// TIA Portal project "2022.09.06-步进电机仿真" (V17)

(* hardware
DEVICE "HMI_1"  KTP700 Basic PN
   slot 0: "HMI_1"  KTP700 Basic PN  6AV2 123-2GB03-0AX0  15.1.0.0
   slot 1: "HMI_RT_1"  KTP700 Basic PN  6AV2 123-2GB03-0AX0  15.1.0.0
   slot 5: "HMI_1.IE_CP_1"  PROFINET Interface  15.0.1.0
      slot 1: "PROFINET Interface_1"  PROFINET Interface
         slot 1: "Port_1"  Port
DEVICE "S7-1200 station_1"  S7-1200 Station
   slot 0: "Rack_0"  S7-1200 Rack  Rack  V1.0
   slot 1: "PLC_1"  CPU 1214C DC/DC/DC  6ES7 214-1AG40-0XB0  V4.2
*)

// ===== PLC "PLC_1"  CPU 1214C DC/DC/DC =====

VAR_GLOBAL   // PLC tag table "默认变量表"
   "反转按钮" AT %I0.1 : Bool;
   "正转KA1" AT %Q0.0 : Bool;
   "反转KA2" AT %Q0.1 : Bool;
   "停止按钮" AT %I0.2 : Bool;
   "正转按钮" AT %I0.0 : Bool;
   "正转按钮触摸屏" AT %M0.0 : Bool;
   "反转按钮触摸屏" AT %M0.1 : Bool;
   "停止按钮触摸屏" AT %M0.2 : Bool;
   "正转触摸屏指示灯" AT %M1.0 : Bool;
   "反转触摸屏指示灯" AT %M1.1 : Bool;
   "电动机转速" AT %MD20 : DWord;
END_VAR

ORGANIZATION_BLOCK "Main"   // OB1, LAD, ProgramCycle
TITLE = "Main Program Sweep (Cycle)"
{ S7_Optimized_Access := 'TRUE' }
VERSION : 0.1
   VAR_INPUT
      Initial_Call : Bool;   // Initial call of this OB
      Remanence : Bool;   // =True, if remanent data are available
   END_VAR
BEGIN

REGION Network 1
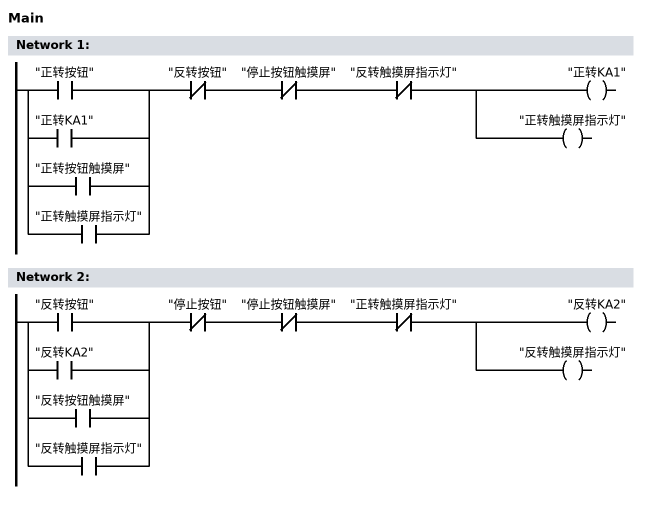
   RUNG wire#powerrail
      Contact( "正转按钮" )
      wire#w1
      I_Contact( "反转按钮" )
      I_Contact( "停止按钮触摸屏" )
      I_Contact( "反转触摸屏指示灯" )
      wire#w2
      Coil( "正转KA1" )
   END_RUNG
   RUNG wire#powerrail
      Contact( "正转KA1" )
   END_RUNG wire#w1
   RUNG wire#powerrail
      Contact( "正转按钮触摸屏" )
   END_RUNG wire#w1
   RUNG wire#powerrail
      Contact( "正转触摸屏指示灯" )
   END_RUNG wire#w1
   RUNG wire#w2
      Coil( "正转触摸屏指示灯" )
   END_RUNG
   // the same network as SCL:
   "正转KA1" := ("正转按钮" OR "正转KA1" OR "正转按钮触摸屏" OR "正转触摸屏指示灯") AND NOT "反转按钮" AND NOT "停止按钮触摸屏" AND NOT "反转触摸屏指示灯";
   "正转触摸屏指示灯" := "正转KA1";
END_REGION

REGION Network 2
   RUNG wire#powerrail
      Contact( "反转按钮" )
      wire#w1
      I_Contact( "停止按钮" )
      I_Contact( "停止按钮触摸屏" )
      I_Contact( "正转触摸屏指示灯" )
      wire#w2
      Coil( "反转KA2" )
   END_RUNG
   RUNG wire#powerrail
      Contact( "反转KA2" )
   END_RUNG wire#w1
   RUNG wire#powerrail
      Contact( "反转按钮触摸屏" )
   END_RUNG wire#w1
   RUNG wire#powerrail
      Contact( "反转触摸屏指示灯" )
   END_RUNG wire#w1
   RUNG wire#w2
      Coil( "反转触摸屏指示灯" )
   END_RUNG
   // the same network as SCL:
   "反转KA2" := ("反转按钮" OR "反转KA2" OR "反转按钮触摸屏" OR "反转触摸屏指示灯") AND NOT "停止按钮" AND NOT "停止按钮触摸屏" AND NOT "正转触摸屏指示灯";
   "反转触摸屏指示灯" := "反转KA2";
END_REGION
END_ORGANIZATION_BLOCK

(* ===== HMI "HMI_RT_1" =====
system functions are stored by id; their names below are inferred from use
connection "HMI_连接_1": ETHERNET, SMART_S7_1200_OMS

HMI tags "默认变量表"
   "正转按钮触摸屏" : Bool = PLC 正转按钮触摸屏 AT %M0.0, 1 s
   "反转按钮触摸屏" : Bool = PLC 反转按钮触摸屏 AT %M0.1, 1 s
   "停止按钮触摸屏" : Bool = PLC 停止按钮触摸屏 AT %M0.2, 1 s
   "正转触摸屏指示灯" : Bool = PLC 正转触摸屏指示灯 AT %M1.0, 1 s
   "反转触摸屏指示灯" : Bool = PLC 反转触摸屏指示灯 AT %M1.1, 1 s
   "电动机转速" : DWord = PLC 电动机转速 AT %MD20, 1 s

screen "画面_1" 800x480
   Button "按钮_1" at 140,122 size 104x35; TextOff '正转按钮'
      on Press: SetBit("正转按钮触摸屏")
      on Release: ResetBit("正转按钮触摸屏")
   Button "按钮_2" at 140,199 size 104x35; TextOff '反转按钮'
      on Press: SetBit("反转按钮触摸屏")
      on Release: ResetBit("反转按钮触摸屏")
   Button "按钮_3" at 140,270 size 104x35; TextOff '停止按钮'
      on Press: SetBit("停止按钮触摸屏")
      on Release: ResetBit("停止按钮触摸屏")
   Circle "圆_1" at 428,186 size 48x48
      Appearance <- "正转触摸屏指示灯"
   Circle "圆_2" at 429,263 size 48x48
      Appearance <- "反转触摸屏指示灯"
   TextField "文本域_1" at 521,199 size 125x27; Text '正转指示灯'
   TextField "文本域_2" at 519,276 size 125x27; Text '反转指示灯'
   TextField "文本域_3" at 209,30 size 449x40; Text '直流电机正反转及调速控制'
   IOField "I/O 域_1" at 397,124 size 96x32; FormatPattern 999
      ProcessValue <- "电动机转速"
   TextField "文本域_4" at 519,127 size 125x27; Text '电动机调速'
*)